(* CoDeSys 2.3 export: SCENE.EXP *)

(* POU Components/Scene/Scene, ST *)
FUNCTION_BLOCK Scene
VAR_INPUT
	rotate:BOOL;
	switch:BOOL;
END_VAR

VAR
	count:INT:=3;
	number:INT;
	enabled:BOOL;
	privateNumber:INT;
END_VAR
enabled:= enabled XOR switch;

IF rotate AND enabled THEN
	privateNumber := privateNumber + 1;
END_IF

IF privateNumber >= count OR privateNumber < 1 THEN
	privateNumber:=1;
END_IF

IF enabled THEN
	number := privateNumber;
ELSE
	number := 0;
END_IF
END_FUNCTION_BLOCK
